(*
SPDX-FileCopyrightText: © 2026 Oleksandr Tiutyk <trofimich@gmail.com>
SPDX-License-Identifier: MIT
License: https://opensource.org/license/mit
*)

{attribute 'no_explicit_call' := 'do not call this function block directly'} 
FUNCTION_BLOCK GENERIC_VALUE
VAR_OUTPUT
	TypeClass : GENERIC_TYPE_CLASS;
	Address : POINTER TO BYTE;
	Size : ULINT;
	IsMemoryOwner : BOOL;
END_VAR

METHOD AsAnyType : __SYSTEM.AnyType
AsAnyType := SystemAnyTypes.CreateAnyTypeByGenericValue(THIS^);
END_METHOD

METHOD AsBool : BOOL
VAR
	conversionException : GenericConversionNotSupportedException;
	universalPointer : UNIVERSAL_POINTER;
END_VAR
universalPointer.AsByte := Address;

CASE TypeClass OF
	GENERIC_TYPE_CLASS.BOOLEAN, 
    GENERIC_TYPE_CLASS.INT_8, GENERIC_TYPE_CLASS.INT_16, GENERIC_TYPE_CLASS.INT_32, GENERIC_TYPE_CLASS.INT_64,
    GENERIC_TYPE_CLASS.UINT_8, GENERIC_TYPE_CLASS.UINT_16, GENERIC_TYPE_CLASS.UINT_32, GENERIC_TYPE_CLASS.UINT_64:
		AsBool := universalPointer.AsBool^;
		RETURN;
END_CASE

conversionException.Throw(NamespaceName, ClassName, __POUNAME(), __POSITION(), TypeClass, GENERIC_TYPE_CLASS.BOOLEAN);
END_METHOD

METHOD AsByte : BYTE
VAR_INPUT
	allowTypeCastWithDataLoss : BOOL := FALSE;
END_VAR
VAR
	conversionException : GenericConversionNotSupportedException;
	universalPointer : UNIVERSAL_POINTER;
END_VAR
universalPointer.AsByte := Address;

CASE TypeClass OF
	GENERIC_TYPE_CLASS.BOOLEAN, GENERIC_TYPE_CLASS.UINT_8:
		 AsByte := universalPointer.AsByte^;
		 RETURN;
END_CASE

IF allowTypeCastWithDataLoss THEN
	CASE TypeClass OF
		GENERIC_TYPE_CLASS.UINT_16:
			 AsByte := TO_BYTE(universalPointer.AsWord^);
			 RETURN;
	 
		GENERIC_TYPE_CLASS.UINT_32: 
			 AsByte := TO_BYTE(universalPointer.AsDWord^);
			 RETURN;
	
		GENERIC_TYPE_CLASS.UINT_64:	
			 AsByte := TO_BYTE(universalPointer.AsLWord^);
			 RETURN;
		
		GENERIC_TYPE_CLASS.INT_8: 
			 AsByte := TO_BYTE(universalPointer.AsSInt^);
			 RETURN;
			 
		GENERIC_TYPE_CLASS.INT_16: 
			 AsByte := TO_BYTE(universalPointer.AsInt^);
			 RETURN;
			 
		GENERIC_TYPE_CLASS.INT_32: 
			 AsByte := TO_BYTE(universalPointer.AsDInt^);
			 RETURN;
			 
		GENERIC_TYPE_CLASS.INT_64:
			 AsByte := TO_BYTE(universalPointer.AsLInt^);
			 RETURN;
	END_CASE
END_IF

conversionException.Throw(NamespaceName, ClassName, __POUNAME(), __POSITION(), TypeClass, GENERIC_TYPE_CLASS.UINT_8);
END_METHOD

METHOD AsDate : DATE
VAR_INPUT
	allowTypeCastWithDataLoss : BOOL := FALSE;
END_VAR
VAR
	conversionException : GenericConversionNotSupportedException;
	universalPointer : UNIVERSAL_POINTER;
END_VAR
universalPointer.AsByte := Address;

CASE TypeClass OF
	GENERIC_TYPE_CLASS.DATE_32: 
		 AsDate := universalPointer.AsDate^;
		 RETURN;		 

	GENERIC_TYPE_CLASS.INT_32, GENERIC_TYPE_CLASS.UINT_32: 
		 AsDate := universalPointer.AsDate^;
		 RETURN;		 

	GENERIC_TYPE_CLASS.DATE_AND_TIME_32:
		 AsDate := TO_DATE(universalPointer.AsDateAndTime^);
		 RETURN;
END_CASE

IF allowTypeCastWithDataLoss THEN
	CASE TypeClass OF		 
		GENERIC_TYPE_CLASS.DATE_64:
			 AsDate := TO_DATE(universalPointer.AsLDate^);
			 RETURN;

		GENERIC_TYPE_CLASS.INT_64, GENERIC_TYPE_CLASS.UINT_64:
			 AsDate := TO_DATE(universalPointer.AsULInt^);
			 RETURN;
	END_CASE
END_IF

conversionException.Throw(NamespaceName, ClassName, __POUNAME(), __POSITION(), TypeClass, GENERIC_TYPE_CLASS.DATE_32);
END_METHOD

METHOD AsDateAndTime : DATE_AND_TIME
VAR_INPUT
	allowTypeCastWithDataLoss : BOOL := FALSE;
END_VAR
VAR
	conversionException : GenericConversionNotSupportedException;
	universalPointer : UNIVERSAL_POINTER;
END_VAR
universalPointer.AsByte := Address;

CASE TypeClass OF
	GENERIC_TYPE_CLASS.DATE_AND_TIME_32:
		 AsDateAndTime := universalPointer.AsDateAndTime^;
		 RETURN;

	GENERIC_TYPE_CLASS.INT_32, GENERIC_TYPE_CLASS.UINT_32:
		 AsDateAndTime := TO_DT(universalPointer.AsUDInt^);
		 RETURN;
		
	GENERIC_TYPE_CLASS.DATE_32:
		 AsDateAndTime := TO_DT(universalPointer.AsDate^);
		 RETURN;
END_CASE

IF allowTypeCastWithDataLoss THEN
	CASE TypeClass OF		 
		GENERIC_TYPE_CLASS.DATE_AND_TIME_64:
			 AsDateAndTime := TO_DT(universalPointer.AsLDateAndTime^);
			 RETURN;

		GENERIC_TYPE_CLASS.INT_64, GENERIC_TYPE_CLASS.UINT_64:
			 AsDateAndTime := TO_DT(universalPointer.AsULInt^);
			 RETURN;
	END_CASE
END_IF

conversionException.Throw(NamespaceName, ClassName, __POUNAME(), __POSITION(), TypeClass, GENERIC_TYPE_CLASS.DATE_AND_TIME_32);
END_METHOD

METHOD AsDInt : DINT
VAR_INPUT
	allowTypeCastWithDataLoss : BOOL := FALSE;
END_VAR
VAR
	conversionException : GenericConversionNotSupportedException;
	universalPointer : UNIVERSAL_POINTER;
END_VAR
universalPointer.AsByte := Address;

CASE TypeClass OF
	GENERIC_TYPE_CLASS.BOOLEAN, GENERIC_TYPE_CLASS.UINT_8:
		 AsDInt := TO_DINT(universalPointer.AsByte^);
		 RETURN;
		
	GENERIC_TYPE_CLASS.UINT_16:
		 AsDInt := TO_DINT(universalPointer.AsWord^);
		 RETURN;

	GENERIC_TYPE_CLASS.INT_8: 
		 AsDInt := TO_DINT(universalPointer.AsSInt^);
		 RETURN;
		 
	GENERIC_TYPE_CLASS.INT_16: 
		 AsDInt := TO_DINT(universalPointer.AsInt^);
		 RETURN;
		 
	GENERIC_TYPE_CLASS.INT_32: 
		 AsDInt := universalPointer.AsDInt^;
		 RETURN;
END_CASE

IF allowTypeCastWithDataLoss THEN
	CASE TypeClass OF		 
		GENERIC_TYPE_CLASS.UINT_32: 
			 AsDInt := TO_DINT(universalPointer.AsDWord^);
			 RETURN;

		GENERIC_TYPE_CLASS.UINT_64:	
			 AsDInt := TO_DINT(universalPointer.AsLWord^);
			 RETURN;
			 			 
		GENERIC_TYPE_CLASS.INT_64:
			 AsDInt := TO_DINT(universalPointer.AsLInt^);
			 RETURN;
	END_CASE
END_IF

conversionException.Throw(NamespaceName, ClassName, __POUNAME(), __POSITION(), TypeClass, GENERIC_TYPE_CLASS.INT_32);
END_METHOD

METHOD AsDWord : DWORD
VAR_INPUT
	allowTypeCastWithDataLoss : BOOL := FALSE;
END_VAR
VAR
	conversionException : GenericConversionNotSupportedException;
	universalPointer : UNIVERSAL_POINTER;
END_VAR
universalPointer.AsByte := Address;

CASE TypeClass OF
	GENERIC_TYPE_CLASS.BOOLEAN, GENERIC_TYPE_CLASS.UINT_8:
		 AsDWord := TO_DWORD(universalPointer.AsByte^);
		 RETURN;
		 
	GENERIC_TYPE_CLASS.UINT_16:
		 AsDWord := TO_DWORD(universalPointer.AsWord^);
		 RETURN;
 
	GENERIC_TYPE_CLASS.UINT_32: 
		 AsDWord := universalPointer.AsDWord^;
		 RETURN;
END_CASE

IF allowTypeCastWithDataLoss THEN
	CASE TypeClass OF	
		GENERIC_TYPE_CLASS.UINT_64:	
			 AsDWord := TO_DWORD(universalPointer.AsLWord^);
			 RETURN;
		
		GENERIC_TYPE_CLASS.INT_8: 
			 AsDWord := TO_DWORD(universalPointer.AsSInt^);
			 RETURN;
			 
		GENERIC_TYPE_CLASS.INT_16: 
			 AsDWord := TO_DWORD(universalPointer.AsInt^);
			 RETURN;
			 
		GENERIC_TYPE_CLASS.INT_32: 
			 AsDWord := TO_DWORD(universalPointer.AsDInt^);
			 RETURN;
			 
		GENERIC_TYPE_CLASS.INT_64:
			 AsDWord := TO_DWORD(universalPointer.AsLInt^);
			 RETURN;
	END_CASE
END_IF

conversionException.Throw(NamespaceName, ClassName, __POUNAME(), __POSITION(), TypeClass, GENERIC_TYPE_CLASS.UINT_32);
END_METHOD

METHOD AsInt : INT
VAR_INPUT
	allowTypeCastWithDataLoss : BOOL := FALSE;
END_VAR
VAR
	conversionException : GenericConversionNotSupportedException;
	universalPointer : UNIVERSAL_POINTER;
END_VAR
universalPointer.AsByte := Address;

CASE TypeClass OF
	GENERIC_TYPE_CLASS.BOOLEAN, GENERIC_TYPE_CLASS.UINT_8:
		 AsInt := TO_INT(universalPointer.AsByte^);
		 RETURN;

	GENERIC_TYPE_CLASS.INT_8: 
		 AsInt := TO_INT(universalPointer.AsSInt^);
		 RETURN;
			 
	GENERIC_TYPE_CLASS.INT_16: 
		 AsInt := universalPointer.AsInt^;
		 RETURN;		 
END_CASE

IF allowTypeCastWithDataLoss THEN
	CASE TypeClass OF	 
		GENERIC_TYPE_CLASS.UINT_16:
			 AsInt := TO_INT(universalPointer.AsWord^);
			 RETURN;
			 
		GENERIC_TYPE_CLASS.UINT_32: 
			 AsInt := TO_INT(universalPointer.AsDWord^);
			 RETURN;
	
		GENERIC_TYPE_CLASS.UINT_64:	
			 AsInt := TO_INT(universalPointer.AsLWord^);
			 RETURN;
					 
		GENERIC_TYPE_CLASS.INT_32: 
			 AsInt := TO_INT(universalPointer.AsDInt^);
			 RETURN;
			 
		GENERIC_TYPE_CLASS.INT_64:
			 AsInt := TO_INT(universalPointer.AsLInt^);
			 RETURN;
	END_CASE
END_IF

conversionException.Throw(NamespaceName, ClassName, __POUNAME(), __POSITION(), TypeClass, GENERIC_TYPE_CLASS.INT_16);
END_METHOD

METHOD AsIObject : IObject
VAR
	objectPointer : POINTER TO Object;

	conversionException : GenericConversionNotSupportedException;
END_VAR
IF TypeClass = GENERIC_TYPE_CLASS.OBJECT THEN
	objectPointer := Address;
	
	IF objectPointer <> 0 THEN
		__QUERYINTERFACE(objectPointer^, AsIObject);						
	END_IF
ELSE	
	conversionException.Throw(NamespaceName, ClassName, __POUNAME(), __POSITION(), TypeClass, GENERIC_TYPE_CLASS.OBJECT);		
END_IF
END_METHOD

METHOD AsLDate : LDATE
VAR_INPUT
	allowTypeCastWithDataLoss : BOOL := FALSE;
END_VAR
VAR
	conversionException : GenericConversionNotSupportedException;
	universalPointer : UNIVERSAL_POINTER;
END_VAR
universalPointer.AsByte := Address;

CASE TypeClass OF
	GENERIC_TYPE_CLASS.DATE_64: 
		 AsLDate := universalPointer.AsLDate^;
		 RETURN;		 

	GENERIC_TYPE_CLASS.DATE_32: 
		 AsLDate := TO_LDATE(universalPointer.AsDate^);
		 RETURN;		 
		 
 	GENERIC_TYPE_CLASS.UINT_64, GENERIC_TYPE_CLASS.INT_64: 
		 AsLDate := TO_LDATE(universalPointer.AsULInt^);
		 RETURN;		 

	GENERIC_TYPE_CLASS.DATE_AND_TIME_32: 
		 AsLDate := TO_LDATE(universalPointer.AsDateAndTime^);
		 RETURN;		 
END_CASE

IF allowTypeCastWithDataLoss THEN
	CASE TypeClass OF		 
		GENERIC_TYPE_CLASS.DATE_AND_TIME_64: 
			 AsLDate := TO_LDATE(universalPointer.AsLDateAndTime^);
			 RETURN;		 
	END_CASE
END_IF

conversionException.Throw(NamespaceName, ClassName, __POUNAME(), __POSITION(), TypeClass, GENERIC_TYPE_CLASS.DATE_32);
END_METHOD

METHOD AsLDateAndTime : LDATE_AND_TIME
VAR_INPUT
	allowTypeCastWithDataLoss : BOOL := FALSE;
END_VAR
VAR
	conversionException : GenericConversionNotSupportedException;
	universalPointer : UNIVERSAL_POINTER;
END_VAR
universalPointer.AsByte := Address;

CASE TypeClass OF
	GENERIC_TYPE_CLASS.DATE_AND_TIME_64: 
		 AsLDateAndTime := universalPointer.AsLDateAndTime^;
		 RETURN;		 

	GENERIC_TYPE_CLASS.DATE_AND_TIME_32:
		 AsLDateAndTime := TO_LDT(universalPointer.AsDateAndTime^);
		 RETURN;
		 
	GENERIC_TYPE_CLASS.UINT_64, GENERIC_TYPE_CLASS.INT_64: 
		 AsLDateAndTime := TO_LDT(universalPointer.AsULInt^);
		 RETURN;		 

	GENERIC_TYPE_CLASS.DATE_32:
		 AsLDateAndTime := TO_LDT(universalPointer.AsDate^);
		 RETURN;

	GENERIC_TYPE_CLASS.TIME_32:
		 AsLDateAndTime := TO_LDT(universalPointer.AsTime^);
		 RETURN;
END_CASE

IF allowTypeCastWithDataLoss THEN
	CASE TypeClass OF		 
		GENERIC_TYPE_CLASS.DATE_64: 
			 AsLDateAndTime := TO_LDT(universalPointer.AsLDate^);
			 RETURN;		 

		GENERIC_TYPE_CLASS.TIME_64: 
			 AsLDateAndTime := TO_LDT(universalPointer.AsLTime^);
			 RETURN;		 
	END_CASE
END_IF

conversionException.Throw(NamespaceName, ClassName, __POUNAME(), __POSITION(), TypeClass, GENERIC_TYPE_CLASS.DATE_AND_TIME_32);
END_METHOD

METHOD AsLInt : LINT
VAR_INPUT
	allowTypeCastWithDataLoss : BOOL := FALSE;
END_VAR
VAR
	conversionException : GenericConversionNotSupportedException;
	universalPointer : UNIVERSAL_POINTER;
END_VAR
universalPointer.AsByte := Address;

CASE TypeClass OF
	GENERIC_TYPE_CLASS.BOOLEAN, GENERIC_TYPE_CLASS.UINT_8:
		 AsLInt := TO_LINT(universalPointer.AsByte^);
		 RETURN;
		
	GENERIC_TYPE_CLASS.UINT_16:
		 AsLInt := TO_LINT(universalPointer.AsWord^);
		 RETURN;

	GENERIC_TYPE_CLASS.UINT_32: 
		 AsLInt := TO_LINT(universalPointer.AsDWord^);
		 RETURN;

	GENERIC_TYPE_CLASS.INT_8: 
		 AsLInt := TO_LINT(universalPointer.AsSInt^);
		 RETURN;
		 
	GENERIC_TYPE_CLASS.INT_16: 
		 AsLInt := TO_LINT(universalPointer.AsInt^);
		 RETURN;
		 
	GENERIC_TYPE_CLASS.INT_32: 
		 AsLInt := TO_LINT(universalPointer.AsDInt^);
		 RETURN;
			 			 
	GENERIC_TYPE_CLASS.INT_64:
		 AsLInt := universalPointer.AsLInt^;
		 RETURN;
END_CASE

IF allowTypeCastWithDataLoss THEN
	CASE TypeClass OF		 
		GENERIC_TYPE_CLASS.UINT_64:	
			 AsLInt := TO_LINT(universalPointer.AsLWord^);
			 RETURN;
	END_CASE
END_IF

conversionException.Throw(NamespaceName, ClassName, __POUNAME(), __POSITION(), TypeClass, GENERIC_TYPE_CLASS.INT_64);
END_METHOD

METHOD AsLReal : LREAL
VAR
	conversionException : GenericConversionNotSupportedException;
	universalPointer : UNIVERSAL_POINTER;
END_VAR
universalPointer.AsByte := Address;

CASE TypeClass OF
	GENERIC_TYPE_CLASS.REAL_32:
		 AsLReal := TO_LREAL(universalPointer.AsReal^);
		 RETURN;
	 
	GENERIC_TYPE_CLASS.REAL_64:	
		 AsLReal := universalPointer.AsLReal^;
		 RETURN;
END_CASE

conversionException.Throw(NamespaceName, ClassName, __POUNAME(), __POSITION(), TypeClass, GENERIC_TYPE_CLASS.REAL_64);
END_METHOD

METHOD AsLTime : LTIME
VAR_INPUT
	allowTypeCastWithDataLoss : BOOL := FALSE;
END_VAR
VAR
	conversionException : GenericConversionNotSupportedException;
	universalPointer : UNIVERSAL_POINTER;
END_VAR
universalPointer.AsByte := Address;

CASE TypeClass OF
	GENERIC_TYPE_CLASS.TIME_64:
		 AsLTime := universalPointer.AsLTime^;
		 RETURN;

	GENERIC_TYPE_CLASS.TIME_32: 
		 AsLTime := TO_LTIME(universalPointer.AsTime^);
		 RETURN;
		
	GENERIC_TYPE_CLASS.UINT_64, GENERIC_TYPE_CLASS.INT_64:
		 AsLTime := TO_LTIME(universalPointer.AsULInt^);
		 RETURN;

	GENERIC_TYPE_CLASS.DATE_AND_TIME_32:
		 AsLTime := TO_LTIME(universalPointer.AsDateAndTime^);
		 RETURN;
		 
	GENERIC_TYPE_CLASS.TIME_OF_DAY_32: 
		 AsLTime := TO_LTIME(universalPointer.AsTimeOfDay^);
		 RETURN;
END_CASE

IF allowTypeCastWithDataLoss THEN
	CASE TypeClass OF		 
		GENERIC_TYPE_CLASS.DATE_AND_TIME_64: 
			 AsLTime := TO_LTIME(universalPointer.AsLDateAndTime^);
			 RETURN;		  

		GENERIC_TYPE_CLASS.TIME_OF_DAY_64: 
			 AsLTime := TO_LTIME(universalPointer.AsLTimeOfDay^);
			 RETURN;
	END_CASE
END_IF

conversionException.Throw(NamespaceName, ClassName, __POUNAME(), __POSITION(), TypeClass, GENERIC_TYPE_CLASS.TIME_64);
END_METHOD

METHOD AsLTimeOfDay : LTIME_OF_DAY
VAR_INPUT
	allowTypeCastWithDataLoss : BOOL := FALSE;
END_VAR
VAR
	conversionException : GenericConversionNotSupportedException;
	universalPointer : UNIVERSAL_POINTER;
END_VAR
universalPointer.AsByte := Address;

CASE TypeClass OF
	GENERIC_TYPE_CLASS.TIME_OF_DAY_64: 
		 AsLTimeOfDay := universalPointer.AsLTimeOfDay^;
		 RETURN;

	GENERIC_TYPE_CLASS.TIME_OF_DAY_32: 
		 AsLTimeOfDay :=  TO_LTOD(universalPointer.AsTimeOfDay^);
		 RETURN;

	GENERIC_TYPE_CLASS.UINT_64, GENERIC_TYPE_CLASS.INT_64: 
		 AsLTimeOfDay := TO_LTOD(universalPointer.AsULInt^);
		 RETURN;
		 
	GENERIC_TYPE_CLASS.TIME_32:
		 AsLTimeOfDay := TO_LTOD(universalPointer.AsTime^);
		 RETURN;		 

	GENERIC_TYPE_CLASS.DATE_AND_TIME_32:
		 AsLTimeOfDay := TO_LTOD(universalPointer.AsDateAndTime^);
		 RETURN;		 
END_CASE

IF allowTypeCastWithDataLoss THEN
	CASE TypeClass OF			 
		GENERIC_TYPE_CLASS.TIME_64:
			 AsLTimeOfDay := TO_LTOD(universalPointer.AsLTime^);
			 RETURN;
			 
		GENERIC_TYPE_CLASS.DATE_AND_TIME_64:
			 AsLTimeOfDay := TO_LTOD(universalPointer.AsLDateAndTime^);
			 RETURN;
	END_CASE
END_IF

conversionException.Throw(NamespaceName, ClassName, __POUNAME(), __POSITION(), TypeClass, GENERIC_TYPE_CLASS.TIME_OF_DAY_32);
END_METHOD

METHOD AsLWord : LWORD
VAR_INPUT
	allowTypeCastWithDataLoss : BOOL := FALSE;
END_VAR
VAR
	conversionException : GenericConversionNotSupportedException;
	universalPointer : UNIVERSAL_POINTER;
END_VAR
universalPointer.AsByte := Address;

CASE TypeClass OF
	GENERIC_TYPE_CLASS.BOOLEAN, GENERIC_TYPE_CLASS.UINT_8:
		 AsLWord := TO_LWORD(universalPointer.AsByte^);
		 RETURN;
		 
	GENERIC_TYPE_CLASS.UINT_16:
		 AsLWord := TO_LWORD(universalPointer.AsWord^);
		 RETURN;
 
	GENERIC_TYPE_CLASS.UINT_32: 
		 AsLWord := TO_LWORD(universalPointer.AsDWord^);
		 RETURN;
		 
	GENERIC_TYPE_CLASS.UINT_64:	
		 AsLWord := universalPointer.AsLWord^;
		 RETURN;		 
END_CASE

IF allowTypeCastWithDataLoss THEN
	CASE TypeClass OF			
		GENERIC_TYPE_CLASS.INT_8: 
			 AsLWord := TO_LWORD(universalPointer.AsSInt^);
			 RETURN;
			 
		GENERIC_TYPE_CLASS.INT_16: 
			 AsLWord := TO_LWORD(universalPointer.AsInt^);
			 RETURN;
			 
		GENERIC_TYPE_CLASS.INT_32: 
			 AsLWord := TO_LWORD(universalPointer.AsDInt^);
			 RETURN;
			 
		GENERIC_TYPE_CLASS.INT_64:
			 AsLWord := TO_LWORD(universalPointer.AsLInt^);
			 RETURN;
	END_CASE
END_IF

conversionException.Throw(NamespaceName, ClassName, __POUNAME(), __POSITION(), TypeClass, GENERIC_TYPE_CLASS.UINT_64);
END_METHOD

METHOD AsObject : REFERENCE TO Object
VAR
	objectPointer : POINTER TO Object;

	conversionException : GenericConversionNotSupportedException;
END_VAR
IF TypeClass = GENERIC_TYPE_CLASS.OBJECT THEN
	objectPointer := Address;
	
	IF objectPointer <> 0 THEN
		AsObject REF= objectPointer^;		
	END_IF
ELSE	
	conversionException.Throw(NamespaceName, ClassName, __POUNAME(), __POSITION(), TypeClass, GENERIC_TYPE_CLASS.OBJECT);		
END_IF
END_METHOD

METHOD AsReal : REAL
VAR_INPUT
	allowTypeCastWithDataLoss : BOOL := FALSE;
END_VAR
VAR
	conversionException : GenericConversionNotSupportedException;
	universalPointer : UNIVERSAL_POINTER;
END_VAR
universalPointer.AsByte := Address;

CASE TypeClass OF
	GENERIC_TYPE_CLASS.REAL_32:
		 AsReal := universalPointer.AsReal^;
		 RETURN;
END_CASE

IF allowTypeCastWithDataLoss THEN
	CASE TypeClass OF		 
		GENERIC_TYPE_CLASS.REAL_64:	
			 AsReal := TO_REAL(universalPointer.AsLWord^);
			 RETURN;
	END_CASE
END_IF

conversionException.Throw(NamespaceName, ClassName, __POUNAME(), __POSITION(), TypeClass, GENERIC_TYPE_CLASS.REAL_32);
END_METHOD

METHOD INTERNAL Assign
VAR_INPUT
	genericTypeClass : GENERIC_TYPE_CLASS;
	address : POINTER TO BYTE;
	size : ULINT;
	isMemoryOwner : BOOL;
END_VAR
VAR
	addressNullException : ArgumentNotSpecifiedException;
END_VAR
IF address = 0 THEN
	addressNullException.Throw(NamespaceName, ClassName, __POUNAME(), __POSITION(), 'address');
END_IF

THIS^.TypeClass := genericTypeClass;
THIS^.Address := address;
THIS^.Size := size;
THIS^.IsMemoryOwner := isMemoryOwner;
END_METHOD

METHOD AsSInt : SINT
VAR_INPUT
	allowTypeCastWithDataLoss : BOOL := FALSE;
END_VAR
VAR
	conversionException : GenericConversionNotSupportedException;
	universalPointer : UNIVERSAL_POINTER;
END_VAR
universalPointer.AsByte := Address;

CASE TypeClass OF
	GENERIC_TYPE_CLASS.INT_8: 
		 AsSInt := universalPointer.AsSInt^;
		 RETURN;
END_CASE

IF allowTypeCastWithDataLoss THEN
	CASE TypeClass OF
		GENERIC_TYPE_CLASS.BOOLEAN, GENERIC_TYPE_CLASS.UINT_8:
			 AsSInt := TO_SINT(universalPointer.AsUSInt^);
			 RETURN;
			 
		GENERIC_TYPE_CLASS.UINT_16:
			 AsSInt := TO_SINT(universalPointer.AsWord^);
			 RETURN;
	 
		GENERIC_TYPE_CLASS.UINT_32: 
			 AsSInt := TO_SINT(universalPointer.AsDWord^);
			 RETURN;
	
		GENERIC_TYPE_CLASS.UINT_64:	
			 AsSInt := TO_SINT(universalPointer.AsLWord^);
			 RETURN;
					 
		GENERIC_TYPE_CLASS.INT_16: 
			 AsSInt := TO_SINT(universalPointer.AsInt^);
			 RETURN;
			 
		GENERIC_TYPE_CLASS.INT_32: 
			 AsSInt := TO_SINT(universalPointer.AsDInt^);
			 RETURN;
			 
		GENERIC_TYPE_CLASS.INT_64:
			 AsSInt := TO_SINT(universalPointer.AsLInt^);
			 RETURN;
	END_CASE
END_IF

conversionException.Throw(NamespaceName, ClassName, __POUNAME(), __POSITION(), TypeClass, GENERIC_TYPE_CLASS.INT_8);
END_METHOD

METHOD AsString255 : STRING(255)
VAR_INPUT
	allowTypeCastWithDataLoss : BOOL := FALSE;
END_VAR
VAR
	conversionException : GenericConversionNotSupportedException;
	universalPointer : UNIVERSAL_POINTER;
END_VAR
universalPointer.AsByte := Address;

CASE TypeClass OF
	GENERIC_TYPE_CLASS.BOOLEAN:
		 AsString255 := TO_STRING(universalPointer.AsBool^);
		 RETURN;
    GENERIC_TYPE_CLASS.INT_8:
		 AsString255 := TO_STRING(universalPointer.AsSInt^);
		 RETURN;
    GENERIC_TYPE_CLASS.INT_16:
		 AsString255 := TO_STRING(universalPointer.AsInt^);
		 RETURN;
    GENERIC_TYPE_CLASS.INT_32:
		 AsString255 := TO_STRING(universalPointer.AsDInt^);
		 RETURN;
    GENERIC_TYPE_CLASS.INT_64:
		 AsString255 := TO_STRING(universalPointer.AsLInt^);
		 RETURN;
    GENERIC_TYPE_CLASS.UINT_8:
		 AsString255 := TO_STRING(universalPointer.AsUSInt^);
		 RETURN;
    GENERIC_TYPE_CLASS.UINT_16:
		 AsString255 := TO_STRING(universalPointer.AsUInt^);
		 RETURN;
    GENERIC_TYPE_CLASS.UINT_32:
		 AsString255 := TO_STRING(universalPointer.AsUDInt^);
		 RETURN;
    GENERIC_TYPE_CLASS.UINT_64:
		 AsString255 := TO_STRING(universalPointer.AsULInt^);
		 RETURN;
    GENERIC_TYPE_CLASS.REAL_32:
		 AsString255 := TO_STRING(universalPointer.AsReal^);
		 RETURN;
    GENERIC_TYPE_CLASS.REAL_64:
		 AsString255 := TO_STRING(universalPointer.AsLReal^);
		 RETURN;
    GENERIC_TYPE_CLASS.STRING_ASCII:
		 AsString255 := universalPointer.AsString^;
		 RETURN;
    GENERIC_TYPE_CLASS.TIME_32:
		 AsString255 := TO_STRING(universalPointer.AsTime^);
		 RETURN;
    GENERIC_TYPE_CLASS.TIME_64:
		 AsString255 := TO_STRING(universalPointer.AsLTime^);
		 RETURN;
    GENERIC_TYPE_CLASS.DATE_32:
		 AsString255 := TO_STRING(universalPointer.AsDate^);
		 RETURN;
    GENERIC_TYPE_CLASS.DATE_64:
		 AsString255 := TO_STRING(universalPointer.AsLDate ^);
		 RETURN;
    GENERIC_TYPE_CLASS.DATE_AND_TIME_32:
		 AsString255 := TO_STRING(universalPointer.AsDateAndTime^);
		 RETURN;
    GENERIC_TYPE_CLASS.DATE_AND_TIME_64:
		 AsString255 := TO_STRING(universalPointer.AsLDateAndTime^);
		 RETURN;
    GENERIC_TYPE_CLASS.TIME_OF_DAY_32:
		 AsString255 := TO_STRING(universalPointer.AsTimeOfDay^);
		 RETURN;
    GENERIC_TYPE_CLASS.TIME_OF_DAY_64:
		 AsString255 := TO_STRING(universalPointer.AsLTimeOfDay^);
		 RETURN;
END_CASE

IF allowTypeCastWithDataLoss THEN
	CASE TypeClass OF	 			 
		GENERIC_TYPE_CLASS.STRING_UTF16:
			 AsString255 := TO_STRING(universalPointer.AsWString^);
			 RETURN;
	END_CASE
END_IF

conversionException.Throw(NamespaceName, ClassName, __POUNAME(), __POSITION(), TypeClass, GENERIC_TYPE_CLASS.STRING_ASCII);
END_METHOD

METHOD AsStringReference : REFERENCE TO STRING
VAR
	conversionException : GenericConversionNotSupportedException;
	universalPointer : UNIVERSAL_POINTER;
END_VAR
universalPointer.AsByte := Address;

CASE TypeClass OF
    GENERIC_TYPE_CLASS.STRING_ASCII:
		 AsStringReference REF= universalPointer.AsString^;
		 RETURN;
END_CASE

conversionException.Throw(NamespaceName, ClassName, __POUNAME(), __POSITION(), TypeClass, GENERIC_TYPE_CLASS.STRING_ASCII);
END_METHOD

METHOD AsTime : TIME
VAR_INPUT
	allowTypeCastWithDataLoss : BOOL := FALSE;
END_VAR
VAR
	conversionException : GenericConversionNotSupportedException;
	universalPointer : UNIVERSAL_POINTER;
END_VAR
universalPointer.AsByte := Address;

CASE TypeClass OF
	GENERIC_TYPE_CLASS.DATE_AND_TIME_32:
		 AsTime := TO_TIME(universalPointer.AsDateAndTime^);
		 RETURN;

	GENERIC_TYPE_CLASS.INT_32, GENERIC_TYPE_CLASS.UINT_32:
		AsTime := TO_TIME(universalPointer.AsUDInt^);
		RETURN;
		
	GENERIC_TYPE_CLASS.TIME_32: 
		 AsTime := universalPointer.AsTime^;
		 RETURN;
		 
	GENERIC_TYPE_CLASS.TIME_OF_DAY_32: 
		 AsTime := TO_TIME(universalPointer.AsTimeOfDay^);
		 RETURN;
END_CASE

IF allowTypeCastWithDataLoss THEN
	CASE TypeClass OF		 
		GENERIC_TYPE_CLASS.TIME_64:
			 AsTime := TO_TIME(universalPointer.AsLTime^);
			 RETURN;

		GENERIC_TYPE_CLASS.INT_64, GENERIC_TYPE_CLASS.UINT_64:
			AsTime := TO_TIME(universalPointer.AsULInt^);
			RETURN;
	END_CASE
END_IF

conversionException.Throw(NamespaceName, ClassName, __POUNAME(), __POSITION(), TypeClass, GENERIC_TYPE_CLASS.TIME_32);
END_METHOD

METHOD AsTimeOfDay : TIME_OF_DAY
VAR_INPUT
	allowTypeCastWithDataLoss : BOOL := FALSE;
END_VAR
VAR
	conversionException : GenericConversionNotSupportedException;
	universalPointer : UNIVERSAL_POINTER;
END_VAR
universalPointer.AsByte := Address;

CASE TypeClass OF
	GENERIC_TYPE_CLASS.TIME_OF_DAY_32: 
		 AsTimeOfDay := universalPointer.AsTimeOfDay^;
		 RETURN;

	GENERIC_TYPE_CLASS.INT_32, GENERIC_TYPE_CLASS.UINT_32: 
		 AsTimeOfDay := TO_TOD(universalPointer.AsUDInt^);
		 RETURN;
END_CASE

IF allowTypeCastWithDataLoss THEN
	CASE TypeClass OF
		GENERIC_TYPE_CLASS.TIME_32:
			 AsTimeOfDay := TO_TOD(universalPointer.AsTime^);
			 RETURN;
	
		GENERIC_TYPE_CLASS.INT_64, GENERIC_TYPE_CLASS.UINT_64: 
			 AsTimeOfDay := TO_TOD(universalPointer.AsULInt^);
			 RETURN;
			 
		GENERIC_TYPE_CLASS.TIME_64:
			 AsTimeOfDay := TO_TOD(universalPointer.AsLTime^);
			 RETURN;
	END_CASE
END_IF

conversionException.Throw(NamespaceName, ClassName, __POUNAME(), __POSITION(), TypeClass, GENERIC_TYPE_CLASS.TIME_OF_DAY_32);
END_METHOD

METHOD AsUDInt : UDINT
VAR_INPUT
	allowTypeCastWithDataLoss : BOOL := FALSE;
END_VAR
VAR
	conversionException : GenericConversionNotSupportedException;
	universalPointer : UNIVERSAL_POINTER;
END_VAR
universalPointer.AsByte := Address;

CASE TypeClass OF
	GENERIC_TYPE_CLASS.BOOLEAN, GENERIC_TYPE_CLASS.UINT_8:
		 AsUDInt := TO_UDINT(universalPointer.AsByte^);
		 RETURN;
		 
	GENERIC_TYPE_CLASS.UINT_16:
		 AsUDInt := TO_UDINT(universalPointer.AsWord^);
		 RETURN;
 
	GENERIC_TYPE_CLASS.UINT_32: 
		 AsUDInt := universalPointer.AsDWord^;
		 RETURN;
END_CASE

IF allowTypeCastWithDataLoss THEN
	CASE TypeClass OF	
		GENERIC_TYPE_CLASS.UINT_64:	
			 AsUDInt := TO_UDINT(universalPointer.AsLWord^);
			 RETURN;
		
		GENERIC_TYPE_CLASS.INT_8: 
			 AsUDInt := TO_UDINT(universalPointer.AsSInt^);
			 RETURN;
			 
		GENERIC_TYPE_CLASS.INT_16: 
			 AsUDInt := TO_UDINT(universalPointer.AsInt^);
			 RETURN;
			 
		GENERIC_TYPE_CLASS.INT_32: 
			 AsUDInt := TO_UDINT(universalPointer.AsDInt^);
			 RETURN;
			 
		GENERIC_TYPE_CLASS.INT_64:
			 AsUDInt := TO_UDINT(universalPointer.AsLInt^);
			 RETURN;
	END_CASE
END_IF

conversionException.Throw(NamespaceName, ClassName, __POUNAME(), __POSITION(), TypeClass, GENERIC_TYPE_CLASS.UINT_32);
END_METHOD

METHOD AsUInt : UINT
VAR_INPUT
	allowTypeCastWithDataLoss : BOOL := FALSE;
END_VAR
VAR
	conversionException : GenericConversionNotSupportedException;
	universalPointer : UNIVERSAL_POINTER;
END_VAR
universalPointer.AsByte := Address;

CASE TypeClass OF
	GENERIC_TYPE_CLASS.BOOLEAN, GENERIC_TYPE_CLASS.UINT_8:
		 AsUInt := TO_UINT(universalPointer.AsByte^);
		 RETURN;
		 
	GENERIC_TYPE_CLASS.UINT_16:
		 AsUInt := universalPointer.AsWord^;
		 RETURN;
END_CASE

IF allowTypeCastWithDataLoss THEN
	CASE TypeClass OF	 
		GENERIC_TYPE_CLASS.UINT_32: 
			 AsUInt := TO_UINT(universalPointer.AsDWord^);
			 RETURN;
	
		GENERIC_TYPE_CLASS.UINT_64:	
			 AsUInt := TO_UINT(universalPointer.AsLWord^);
			 RETURN;
		
		GENERIC_TYPE_CLASS.INT_8: 
			 AsUInt := TO_UINT(universalPointer.AsSInt^);
			 RETURN;
			 
		GENERIC_TYPE_CLASS.INT_16: 
			 AsUInt := TO_UINT(universalPointer.AsInt^);
			 RETURN;
			 
		GENERIC_TYPE_CLASS.INT_32: 
			 AsUInt := TO_UINT(universalPointer.AsDInt^);
			 RETURN;
			 
		GENERIC_TYPE_CLASS.INT_64:
			 AsUInt := TO_UINT(universalPointer.AsLInt^);
			 RETURN;
	END_CASE
END_IF

conversionException.Throw(NamespaceName, ClassName, __POUNAME(), __POSITION(), TypeClass, GENERIC_TYPE_CLASS.UINT_16);
END_METHOD

METHOD AsULInt : ULINT
VAR_INPUT
	allowTypeCastWithDataLoss : BOOL := FALSE;
END_VAR
VAR
	conversionException : GenericConversionNotSupportedException;
	universalPointer : UNIVERSAL_POINTER;
END_VAR
universalPointer.AsByte := Address;

CASE TypeClass OF
	GENERIC_TYPE_CLASS.BOOLEAN, GENERIC_TYPE_CLASS.UINT_8:
		 AsULInt := TO_ULINT(universalPointer.AsByte^);
		 RETURN;
		 
	GENERIC_TYPE_CLASS.UINT_16:
		 AsULInt := TO_ULINT(universalPointer.AsWord^);
		 RETURN;
 
	GENERIC_TYPE_CLASS.UINT_32: 
		 AsULInt := TO_ULINT(universalPointer.AsDWord^);
		 RETURN;
		 
	GENERIC_TYPE_CLASS.UINT_64:	
		 AsULInt := universalPointer.AsLWord^;
		 RETURN;		 
END_CASE

IF allowTypeCastWithDataLoss THEN
	CASE TypeClass OF			
		GENERIC_TYPE_CLASS.INT_8: 
			 AsULInt := TO_ULINT(universalPointer.AsSInt^);
			 RETURN;
			 
		GENERIC_TYPE_CLASS.INT_16: 
			 AsULInt := TO_ULINT(universalPointer.AsInt^);
			 RETURN;
			 
		GENERIC_TYPE_CLASS.INT_32: 
			 AsULInt := TO_ULINT(universalPointer.AsDInt^);
			 RETURN;
			 
		GENERIC_TYPE_CLASS.INT_64:
			 AsULInt := TO_ULINT(universalPointer.AsLInt^);
			 RETURN;
	END_CASE
END_IF

conversionException.Throw(NamespaceName, ClassName, __POUNAME(), __POSITION(), TypeClass, GENERIC_TYPE_CLASS.UINT_64);
END_METHOD

METHOD AsUSInt : USINT
VAR_INPUT
	allowTypeCastWithDataLoss : BOOL := FALSE;
END_VAR
VAR
	conversionException : GenericConversionNotSupportedException;
	universalPointer : UNIVERSAL_POINTER;
END_VAR
universalPointer.AsByte := Address;

CASE TypeClass OF
	GENERIC_TYPE_CLASS.BOOLEAN, GENERIC_TYPE_CLASS.UINT_8:
		 AsUSInt := universalPointer.AsUSInt^;
		 RETURN;
END_CASE

IF allowTypeCastWithDataLoss THEN
	CASE TypeClass OF
		GENERIC_TYPE_CLASS.UINT_16:
			 AsUSInt := TO_USINT(universalPointer.AsWord^);
			 RETURN;
	 
		GENERIC_TYPE_CLASS.UINT_32: 
			 AsUSInt := TO_USINT(universalPointer.AsDWord^);
			 RETURN;
	
		GENERIC_TYPE_CLASS.UINT_64:	
			 AsUSInt := TO_USINT(universalPointer.AsLWord^);
			 RETURN;
		
		GENERIC_TYPE_CLASS.INT_8: 
			 AsUSInt := TO_USINT(universalPointer.AsSInt^);
			 RETURN;
			 
		GENERIC_TYPE_CLASS.INT_16: 
			 AsUSInt := TO_USINT(universalPointer.AsInt^);
			 RETURN;
			 
		GENERIC_TYPE_CLASS.INT_32: 
			 AsUSInt := TO_USINT(universalPointer.AsDInt^);
			 RETURN;
			 
		GENERIC_TYPE_CLASS.INT_64:
			 AsUSInt := TO_USINT(universalPointer.AsLInt^);
			 RETURN;
	END_CASE
END_IF

conversionException.Throw(NamespaceName, ClassName, __POUNAME(), __POSITION(), TypeClass, GENERIC_TYPE_CLASS.UINT_8);
END_METHOD

METHOD AsWord : WORD
VAR_INPUT
	allowTypeCastWithDataLoss : BOOL := FALSE;
END_VAR
VAR
	conversionException : GenericConversionNotSupportedException;
	universalPointer : UNIVERSAL_POINTER;
END_VAR
universalPointer.AsByte := Address;

CASE TypeClass OF
	GENERIC_TYPE_CLASS.BOOLEAN, GENERIC_TYPE_CLASS.UINT_8:
		 AsWord := TO_WORD(universalPointer.AsByte^);
		 RETURN;
		 
	GENERIC_TYPE_CLASS.UINT_16:
		 AsWord := universalPointer.AsWord^;
		 RETURN;
END_CASE

IF allowTypeCastWithDataLoss THEN
	CASE TypeClass OF	 
		GENERIC_TYPE_CLASS.UINT_32: 
			 AsWord := TO_WORD(universalPointer.AsDWord^);
			 RETURN;
	
		GENERIC_TYPE_CLASS.UINT_64:	
			 AsWord := TO_WORD(universalPointer.AsLWord^);
			 RETURN;
		
		GENERIC_TYPE_CLASS.INT_8: 
			 AsWord := TO_WORD(universalPointer.AsSInt^);
			 RETURN;
			 
		GENERIC_TYPE_CLASS.INT_16: 
			 AsWord := TO_WORD(universalPointer.AsInt^);
			 RETURN;
			 
		GENERIC_TYPE_CLASS.INT_32: 
			 AsWord := TO_WORD(universalPointer.AsDInt^);
			 RETURN;
			 
		GENERIC_TYPE_CLASS.INT_64:
			 AsWord := TO_WORD(universalPointer.AsLInt^);
			 RETURN;
	END_CASE
END_IF

conversionException.Throw(NamespaceName, ClassName, __POUNAME(), __POSITION(), TypeClass, GENERIC_TYPE_CLASS.UINT_16);
END_METHOD

METHOD AsWString255 : WSTRING(255)
VAR
	conversionException : GenericConversionNotSupportedException;
	universalPointer : UNIVERSAL_POINTER;
END_VAR
universalPointer.AsByte := Address;

CASE TypeClass OF
	GENERIC_TYPE_CLASS.BOOLEAN:
		 AsWString255 := TO_WSTRING(universalPointer.AsBool^);
		 RETURN;
    GENERIC_TYPE_CLASS.INT_8:
		 AsWString255 := TO_WSTRING(universalPointer.AsSInt^);
		 RETURN;
    GENERIC_TYPE_CLASS.INT_16:
		 AsWString255 := TO_WSTRING(universalPointer.AsInt^);
		 RETURN;
    GENERIC_TYPE_CLASS.INT_32:
		 AsWString255 := TO_WSTRING(universalPointer.AsDInt^);
		 RETURN;
    GENERIC_TYPE_CLASS.INT_64:
		 AsWString255 := TO_WSTRING(universalPointer.AsLInt^);
		 RETURN;
    GENERIC_TYPE_CLASS.UINT_8:
		 AsWString255 := TO_WSTRING(universalPointer.AsUSInt^);
		 RETURN;
    GENERIC_TYPE_CLASS.UINT_16:
		 AsWString255 := TO_WSTRING(universalPointer.AsUInt^);
		 RETURN;
    GENERIC_TYPE_CLASS.UINT_32:
		 AsWString255 := TO_WSTRING(universalPointer.AsUDInt^);
		 RETURN;
    GENERIC_TYPE_CLASS.UINT_64:
		 AsWString255 := TO_WSTRING(universalPointer.AsULInt^);
		 RETURN;
    GENERIC_TYPE_CLASS.REAL_32:
		 AsWString255 := TO_WSTRING(universalPointer.AsReal^);
		 RETURN;
    GENERIC_TYPE_CLASS.REAL_64:
		 AsWString255 := TO_WSTRING(universalPointer.AsLReal^);
		 RETURN;
    GENERIC_TYPE_CLASS.STRING_ASCII:
		 AsWString255 := TO_WSTRING(universalPointer.AsString^);
		 RETURN;
	GENERIC_TYPE_CLASS.STRING_UTF16:
		 AsWString255 := universalPointer.AsWString^;
		 RETURN;
    GENERIC_TYPE_CLASS.TIME_32:
		 AsWString255 := TO_WSTRING(universalPointer.AsTime^);
		 RETURN;
    GENERIC_TYPE_CLASS.TIME_64:
		 AsWString255 := TO_WSTRING(universalPointer.AsLTime^);
		 RETURN;
    GENERIC_TYPE_CLASS.DATE_32:
		 AsWString255 := TO_WSTRING(universalPointer.AsDate^);
		 RETURN;
    GENERIC_TYPE_CLASS.DATE_64:
		 AsWString255 := TO_WSTRING(universalPointer.AsLDate^);
		 RETURN;
    GENERIC_TYPE_CLASS.DATE_AND_TIME_32:
		 AsWString255 := TO_WSTRING(universalPointer.AsDateAndTime^);
		 RETURN;
    GENERIC_TYPE_CLASS.DATE_AND_TIME_64:
		 AsWString255 := TO_WSTRING(universalPointer.AsLDateAndTime^);
		 RETURN;
    GENERIC_TYPE_CLASS.TIME_OF_DAY_32:
		 AsWString255 := TO_WSTRING(universalPointer.AsTimeOfDay^);
		 RETURN;
    GENERIC_TYPE_CLASS.TIME_OF_DAY_64:
		 AsWString255 := TO_WSTRING(universalPointer.AsLTimeOfDay^);
		 RETURN;
END_CASE

conversionException.Throw(NamespaceName, ClassName, __POUNAME(), __POSITION(), TypeClass, GENERIC_TYPE_CLASS.STRING_UTF16);
END_METHOD

METHOD AsWStringReference : REFERENCE TO WSTRING
VAR
	conversionException : GenericConversionNotSupportedException;
	universalPointer : UNIVERSAL_POINTER;
END_VAR
universalPointer.AsByte := Address;

CASE TypeClass OF
	GENERIC_TYPE_CLASS.STRING_UTF16:
		 AsWStringReference REF= universalPointer.AsWString^;
		 RETURN;
END_CASE

conversionException.Throw(NamespaceName, ClassName, __POUNAME(), __POSITION(), TypeClass, GENERIC_TYPE_CLASS.STRING_UTF16);
END_METHOD

METHOD ChangeValueByAny
VAR_INPUT
	value : ANY;
	isObject : BOOL := FALSE;
END_VAR
ChangeValueByAnyType(value, isObject);
END_METHOD

METHOD ChangeValueByAnyType
VAR_INPUT
	value : __SYSTEM.AnyType;
	isObject : BOOL := FALSE;
END_VAR
VAR
	argumentDataType : GENERIC_TYPE_CLASS;
	
	exception : StandardException;
END_VAR
argumentDataType := GenericTypeClassConvertor.GetGenericTypeClassBySystemAnyType(value, isObject);

IF argumentDataType <> TypeClass THEN
	exception.Throw(NamespaceName, ClassName, __POUNAME(), __POSITION(), WideStrings.Concat255("Incompatible argument type '", TO_WSTRING(argumentDataType), "' and generic  type '", TO_WSTRING(TypeClass), "'")); 
END_IF

IF Size < TO_ULINT(value.diSize) THEN
	exception.Throw(NamespaceName, ClassName, __POUNAME(), __POSITION(), WideStrings.Concat255("Insufficient memory size: avaliable - ", TO_WSTRING(Size), ", required - ", TO_WSTRING(value.diSize))); 	
END_IF

IF Tc2_System.MEMCPY(Address, value.pValue, TO_UDINT(value.diSize)) = 0 THEN
	exception.Throw(NamespaceName, ClassName, __POUNAME(), __POSITION(), "Tc2_System.MEMCPY returned error (value 0)"); 		
END_IF
END_METHOD

{attribute 'monitoring' := 'call'}
PROPERTY ClassName : REFERENCE TO STRING
GET
ClassName REF= GenericValueFactory.GenericValueClassName;
END_GET
END_PROPERTY

METHOD CopyTo
VAR_INPUT
	target : ANY;
END_VAR
VAR
	argumentNullException : ArgumentNotSpecifiedException;
	invalidTargetMemorySizeException : StandardException;
END_VAR
IF target.pValue = 0 THEN
	argumentNullException.Throw(NamespaceName, ClassName, __POUNAME(), __POSITION(), 'target'); 
END_IF

IF TO_ULINT(target.diSize) <> Size THEN
	invalidTargetMemorySizeException.Throw(NamespaceName, ClassName, __POUNAME(), __POSITION(), WideStrings.Concat255("Target variable size ", TO_WSTRING(target.diSize), " is not equals to generic variable size ", TO_WSTRING(Size)));
END_IF

internalCopyTo(target.pValue);
END_METHOD

METHOD Equals : BOOL
VAR_INPUT
	otherValue : GENERIC_VALUE;
END_VAR
VAR
	stringPointer : POINTER TO STRING;
	wideStringPointer : POINTER TO WSTRING;
	referenceDataSize : ULINT;
	valueToComapreDataSize : ULINT;
END_VAR
IF Address = 0 OR_ELSE Size = 0 OR_ELSE otherValue.Address = 0 OR_ELSE otherValue.Size = 0 THEN
	Equals := (Address = 0 OR_ELSE Size = 0) AND_THEN (otherValue.Address = 0 OR_ELSE otherValue.Size = 0);
ELSE
	IF TypeClass = GENERIC_TYPE_CLASS.STRING_ASCII AND_THEN otherValue.TypeClass = GENERIC_TYPE_CLASS.STRING_ASCII THEN
		stringPointer := Address;
		referenceDataSize := Strings.GetActualSize(stringPointer^);
		
		stringPointer := otherValue.Address;		
		valueToComapreDataSize := Strings.GetActualSize(stringPointer^);
	ELSIF TypeClass = GENERIC_TYPE_CLASS.STRING_UTF16 AND_THEN otherValue.TypeClass = GENERIC_TYPE_CLASS.STRING_UTF16 THEN
		wideStringPointer := Address;
		referenceDataSize := WideStrings.GetActualSize(wideStringPointer^);
		
		wideStringPointer := otherValue.Address;		
		valueToComapreDataSize := WideStrings.GetActualSize(wideStringPointer^);
	ELSE
		referenceDataSize := Size;
		valueToComapreDataSize := otherValue.Size;		
	END_IF
 
	Equals := referenceDataSize = valueToComapreDataSize AND_THEN Tc2_System.MEMCMP(Address, otherValue.Address, TO_UDINT(referenceDataSize)) = 0;
END_IF
END_METHOD

METHOD PRIVATE internalCopyTo
VAR_INPUT
	targetAddress : PVOID;
END_VAR
IF Address = 0 THEN
	Tc2_System.MEMSET(targetAddress, 0, TO_UDINT(Size));
ELSE
	Tc2_System.MEMCPY(targetAddress, Address, TO_UDINT(Size));
END_IF
END_METHOD

{attribute 'monitoring' := 'call'}
PROPERTY FINAL IsNull : BOOL
GET
IsNull := TypeClass = GENERIC_TYPE_CLASS.UNSPECIFIED OR_ELSE Address = 0 OR_ELSE Size = 0;
END_GET
END_PROPERTY

{attribute 'monitoring' := 'call'}
PROPERTY NamespaceName : REFERENCE TO STRING
GET
NamespaceName REF= CurrentNamespace.Name;
END_GET
END_PROPERTY

METHOD Release
IF IsMemoryOwner THEN
	Memory.TryReleaseDynamicMemory(Address, TypeClass = GENERIC_TYPE_CLASS.OBJECT);
END_IF

Reset();
END_METHOD

METHOD Reset
TypeClass := GENERIC_TYPE_CLASS.UNSPECIFIED;
Address := 0;
Size := 0;
IsMemoryOwner := FALSE;
END_METHOD

METHOD TryChangeValueByAny : BOOL
VAR_INPUT
	value : ANY;
	isObject : BOOL := FALSE;
END_VAR
__TRY
	ChangeValueByAnyType(value, isObject);
	TryChangeValueByAny := TRUE;
__CATCH
__ENDTRY
END_METHOD

METHOD TryChangeValueByAnyType : BOOL
VAR_INPUT
	value : __SYSTEM.AnyType;
	isObject : BOOL := FALSE;
END_VAR
__TRY
	ChangeValueByAnyType(value, isObject);
	TryChangeValueByAnyType := TRUE;
__CATCH
__ENDTRY
END_METHOD

METHOD TryCopyTo : BOOL
VAR_INPUT
	target : ANY;
END_VAR
IF target.pValue = 0 THEN
	RETURN; 
END_IF

IF TO_ULINT(target.diSize) <> Size THEN
	RETURN; 
END_IF

internalCopyTo(target.pValue);

TryCopyTo := TRUE;
END_METHOD

END_FUNCTION_BLOCK

(* stored: Version 1.1.0.1
   POU GENERIC_VALUE: Id {4ec776d3-51b8-42d3-97bb-5e4d1a102b1f}, SpecialFunc None
   Folder AsTyped: Id {e96a41ac-e3cd-4eee-9bfa-b62dba0c2d0e}
   Folder Date and time: Id {0e8135f9-c7a8-41d0-996d-4e135d2a2366}
   Folder Floating point: Id {8039a744-40ce-4546-beea-78a288e45706}
   Folder Integer: Id {e3759741-5c8c-482f-93b9-6ae90a2f6296}
   Folder Signed: Id {fb335c0b-7655-449f-bc46-48fb10ad905c}
   Folder Unsugned: Id {bab4b970-dedd-4b75-8710-280ec540561b}
   Folder Strings: Id {f6373c83-d47f-4dab-9f39-83ae4e8a3796}
   Folder ChangeValue: Id {ff6ec9ec-7e82-4906-a7b3-4f1a0bbc2daf}
   Folder CleanupMethods: Id {6633f1de-b2f9-411c-a1ba-5eaade50e25e}
   Folder Service methods: Id {f60d642b-cec1-4cae-991f-d82121762e9d}
   Method AsAnyType: Id {59db7a53-29a2-4c5e-a06f-b2b343ab8f25}
   Method AsBool: Id {1aaa60f7-a8aa-48fc-a4c3-f53925263a40}
   Method AsByte: Id {936f9e9f-e35c-461b-a5b6-c2e02b118baf}
   Method AsDate: Id {db320a05-493c-45cf-92f8-51bf496ee511}
   Method AsDateAndTime: Id {ba931761-c96e-42e2-9fa4-d1882172beda}
   Method AsDInt: Id {4fea0b7d-fe5e-4808-9a02-b0a72b1114c9}
   Method AsDWord: Id {1ee84003-88d5-466d-8c56-9b5d650c16eb}
   Method AsInt: Id {fbd81b42-6af9-470c-9770-5641903fbac8}
   Method AsIObject: Id {80096a9d-d283-480b-80a4-d0dd536beae0}
   Method AsLDate: Id {a43023c1-e686-4d4d-82c6-573f5b54a6de}
   Method AsLDateAndTime: Id {36a42bba-09cd-44d2-9d6f-f83ecf955631}
   Method AsLInt: Id {557ab87e-2262-4a71-b53a-324d552cca35}
   Method AsLReal: Id {6ff6d2d4-05a2-4a88-8dfa-3efa48fa159c}
   Method AsLTime: Id {312f2003-0852-4cfd-8313-e6043e172de5}
   Method AsLTimeOfDay: Id {3746ef26-79d9-476c-ba8d-9d1fb97744ec}
   Method AsLWord: Id {329d366e-53cb-444a-baae-0e3cbf144975}
   Method AsObject: Id {996e8fad-fcc2-4f05-b582-9a439f872e26}
   Method AsReal: Id {45160cf2-6e60-4035-806b-879e84f1bb89}
   Method Assign: Id {862ebf60-dfb4-45d8-a755-cbc5dc31a2cb}
   Method AsSInt: Id {17b44680-9119-41da-9958-f566e80539b5}
   Method AsString255: Id {34520551-01e7-4ae7-9a34-54ba8a2cf3c1}
   Method AsStringReference: Id {5ecee28b-da1c-4264-92ee-6c69f4328ec9}
   Method AsTime: Id {b0c8a8a8-d7c2-483f-b215-128f7d04ba16}
   Method AsTimeOfDay: Id {83f725a7-471b-4136-801c-36fbe6098098}
   Method AsUDInt: Id {90863b55-b5cf-4472-b2f4-3d7e5196f54f}
   Method AsUInt: Id {0cb7d9b1-a26c-4d44-8107-5807eda8eaa5}
   Method AsULInt: Id {ddfdd7f6-ff0f-4202-a7b9-d1b08069f76c}
   Method AsUSInt: Id {7f2825bd-7342-487e-96ac-27ff3bcc2e3c}
   Method AsWord: Id {5e995462-8574-4174-bafd-d9d8e8e626c5}
   Method AsWString255: Id {02ab723a-3f42-4d36-a0f6-c0e9871bfd09}
   Method AsWStringReference: Id {31493745-1b4b-4427-a5e6-18639dd644fb}
   Method ChangeValueByAny: Id {f7c7dd69-068a-47f7-bb61-709a535f4d37}
   Method ChangeValueByAnyType: Id {1e16a561-f4aa-4df6-80a7-92686d04f493}
   Property ClassName: Id {a1f78ed3-d25a-4e81-8b88-934a58828338}
   Get Get: Id {9652d94e-8909-435e-98b2-6d0f00f73d32}
   Method CopyTo: Id {a9e28a3d-762a-4fcd-99e6-4d377c8be6f0}
   Method Equals: Id {165ded56-3861-403f-9838-406d75321178}
   Method internalCopyTo: Id {dffcbd59-ee39-4c74-bc12-2c951ca57eee}
   Property IsNull: Id {b0a5dbd8-6fb5-436e-9b63-9e18aded8437}
   Get Get: Id {293dd0e0-6dfe-4234-9575-a1a778286228}
   Property NamespaceName: Id {6b1b9ffb-991c-4d04-a51f-7608d3745ab0}
   Get Get: Id {70ea020b-d8b3-4815-b692-efc03598f31f}
   Method Release: Id {9937fc92-8120-434b-ac91-5b20bd6f7de6}
   Method Reset: Id {7b456980-e70d-4684-918f-f6fc89768f34}
   Method TryChangeValueByAny: Id {27b8e08e-2fa6-41be-af60-419256c2188b}
   Method TryChangeValueByAnyType: Id {4ed65d07-87f2-4259-80eb-13281b15e53c}
   Method TryCopyTo: Id {ce4998f1-fc8d-443b-ab31-7fcdb66ae168} *)
